{attribute 'GeneratedUsingTerminal: EL2521-0000-1017'}
{attribute addProperty BoxType "EL2521-0000-1017"}
{attribute addProperty Id "PTO_StatusAT %I*PTO_Status_B24E260C7ENC_Status_compactAT %I*ENC_Status_compact_4C428F887PTO_ControlAT %Q*PTO_Control_9287F8E45PTO_Target_compactAT %Q*PTO_Target_compact_5C359F7D2ENC_Control_compactAT %Q*ENC_Control_compact_2ED727EF3WcStateAT %I*WcState_9091E0EB2InfoDataAT %I*InfoData_94A18F5E2"}
{attribute addProperty CRC "390001265"}
{attribute addProperty Size "28"}
TYPE EL2521_173EF271 EXTENDS EtcSlaveTerminalBase_947E5A46 :
STRUCT
	{attribute addProperty Name "PTO_Status"}
	PTO_Status : PTO_Status_B24E260C;
	{attribute addProperty Name "ENC_Status_compact"}
	ENC_Status_compact : ENC_Status_compact_4C428F88;
	{attribute addProperty Name "PTO_Control"}
	PTO_Control : PTO_Control_9287F8E4;
	{attribute addProperty Name "PTO_Target_compact"}
	PTO_Target_compact : PTO_Target_compact_5C359F7D;
	{attribute addProperty Name "ENC_Control_compact"}
	ENC_Control_compact : ENC_Control_compact_2ED727EF;
	{attribute addProperty Name "WcState"}
	WcState : WcState_9091E0EB;
	{attribute addProperty Name "InfoData"}
	InfoData : InfoData_94A18F5E;
END_STRUCT
END_TYPE

(* stored: Version 1.2.0.0, ProductVersion 3.1.4024.9
   DUT EL2521_173EF271: Id {af0734c2-bd0c-4585-8db1-e7cb99a3733a} *)
